(* PLC project Tc2_Coupler.FB_WriteCouplerRegs Demo, tc3-libraries-kb TwinCAT 3.1 *)
(* stored: creationDateTime 2026-05-10T09:00:00, modificationDateTime 2026-05-10T09:00:00 *)

PROGRAM P_Demo_FB_WriteCouplerRegs
  VAR
    fbFB_WriteCouplerRegs : FB_WriteCouplerRegs;  (* Function blocks 实例 *)
    arg_stState : PLCINTFSTRUCT;  (* VAR_INPUT stState: 2-byte PLC interface 状态字 *)
    arg_nTerminal : BYTE;  (* VAR_INPUT nTerminal: 目标端子号 *)
    arg_nTable : BYTE;  (* VAR_INPUT nTable: 表号 *)
    arg_nStartReg : BYTE;  (* VAR_INPUT nStartReg: 起始寄存器号 *)
    arg_nEndReg : BYTE;  (* VAR_INPUT nEndReg: 结束寄存器号 *)
    arg_bExecute : BOOL;  (* VAR_INPUT bExecute: 上升沿触发 *)
    arg_stCouplerTable : ST_CouplerTable;  (* VAR_INPUT stCouplerTable: 要写入的寄存器值数组 *)
    arg_tTimeout : TIME;  (* VAR_INPUT tTimeout: 执行超时 *)
    out_stCtrl : PLCINTFSTRUCT;  (* VAR_OUTPUT stCtrl: 2-byte PLC interface 控制字 *)
    out_bBusy : BOOL;  (* VAR_OUTPUT bBusy: 执行中 *)
    out_bError : BOOL;  (* VAR_OUTPUT bError: 执行出错 *)
    out_nErrId : UDINT;  (* VAR_OUTPUT nErrId: 错误号 *)
  END_VAR

            // ============================================================
// Tc2_Coupler.FB_WriteCouplerRegs 演示程序
// ============================================================
// 场景：通过 PLC 修改智能端子的标定寄存器（断电后丢失，需用持久存储）
// 验证步骤：
//   1. 引用 Tc2_Coupler（及其依赖：Tc2_System 等）
//   2. 编译 + 登录
//   3. 在线监视各 out_* 输出
//   4. 必要时按场景给 arg_* 输入赋值（详见 doc.md 的'使用注意'）
// ============================================================

fbFB_WriteCouplerRegs(
    stState := arg_stState,
    nTerminal := arg_nTerminal,
    nTable := arg_nTable,
    nStartReg := arg_nStartReg,
    nEndReg := arg_nEndReg,
    bExecute := arg_bExecute,
    stCouplerTable := arg_stCouplerTable,
    tTimeout := arg_tTimeout,
    stCtrl => out_stCtrl,
    bBusy => out_bBusy,
    bError => out_bError,
    nErrId => out_nErrId
);

          
END_PROGRAM
